TYPE CmpConvStopConfig :
STRUCT
	
	HandshakeUpstream: BOOL;
	HasLocate: BOOL; 
	DoesWorkRequest: BOOL;
	HandshakeDownstream: BOOL;
	BufferOnlyOneInMotion: BOOL;
	BufferArrivalFault: BOOL;
	RemoteBufferSensor: BOOL;
	DepartStopFaultTime: TIME;
	TimeSpacingMinimum: TIME;
	BufferArrivalFaultTime: TIME;
	PuckSensorOnTime: TIME;
	PuckSensorOffTime: TIME;
	LocateOpenedSensorOnTime: TIME;
	LocateClosedSensorOnTime: TIME;
	BufferSensorOnTime: TIME;
	BufferSensorOffTime: TIME;

END_STRUCT
END_TYPE

(* stored: Version 1.1.0.1, ProductVersion 3.1.4024.6
   DUT CmpConvStopConfig: Id {490f6674-5985-4496-9990-51a97e9178ec} *)
